ABB RobotStudio station: Tp1_20201210-163829.rsstn

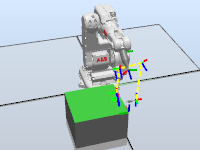
Station Tp1 (saved by RobotStudio 20.2.9116.0)
Controller IRB_140_6kg_0.81m
  mechanical unit ROB_1: IRB140_6_81_C_03, 6 joints, base frame (0, 0, 0) mm
Layout (positions relative to the parent item):
  - IRB140_6_81_C_03 [mechanism, from Robots\IRB140_6_81_C_G_03.rslib] at (0, 0, 0) mm; joint values [0, 0, 0, 3.1416, -0.5236, 3.1416] (rad or m)
  - Mesa [part]
  - Perno [part] at (0, 0, 0) mm
  - Pinza [mechanism] at (506.29, 0, 679.5) mm, rotated rx -180 ry 60 rz -180 deg
      TCP Pinza at (0, 0, 137) mm, rotated rx 0 ry 0 rz -22.5 deg
      links: Dummy
Attachment: Pinza is attached to IRB140_6_81_C_03 / Link6
EventTableEntry 1017: Group=, Trigger=DO_Pinza 1018, Actions=[EventTableActionAttach 1019], Comment=, ActivationMode=2, Cyclic=false
EventTableTriggerIO 1018: IOValue=[1], IRC5Controller=? -1, Operator=0, SignalSource=IRB_140_6kg_0.81m 515
EventTableActionAttach 1019: AttachmentParent=Pinza 1013, AttachmentChild=Perno 1009, MountObject=false, Offset=[X=1, Y=0, Z=0, W=0, X=0, Y=1, Z=0, W=0, X=0, Y=0, Z=1, W=0, X=0, Y=0, Z=0, W=1], FlangeIndext=0, FindNearest=false
EventTableEntry 1020: Group=, Trigger=DO_Pinza 1021, Actions=[EventTableActionDetach 1022], Comment=, ActivationMode=2, Cyclic=false
EventTableTriggerIO 1021: IOValue=[0], IRC5Controller=? -1, Operator=0, SignalSource=IRB_140_6kg_0.81m 515
EventTableActionDetach 1022: AttachmentParent=Pinza 1013, AttachmentChild=Perno 1009
Collision set Colision Perno- Mesa: Perno against Mesa, near miss 0.02 m
Collision set Colision Robot - Mesa: IRB140_6_81_C_03 against Mesa, near miss 0 m
Collision set Colision Pinza - Mesa: Mesa against Pinza, near miss 0 m
EventTableTriggerIO 1093: IOValue=[1], IRC5Controller=? -1, Operator=0, SignalSource=IRB_140_6kg_0.81m 515
EventTableTriggerIO 1094: IOValue=[0], IRC5Controller=? -1, Operator=0, SignalSource=IRB_140_6kg_0.81m 515
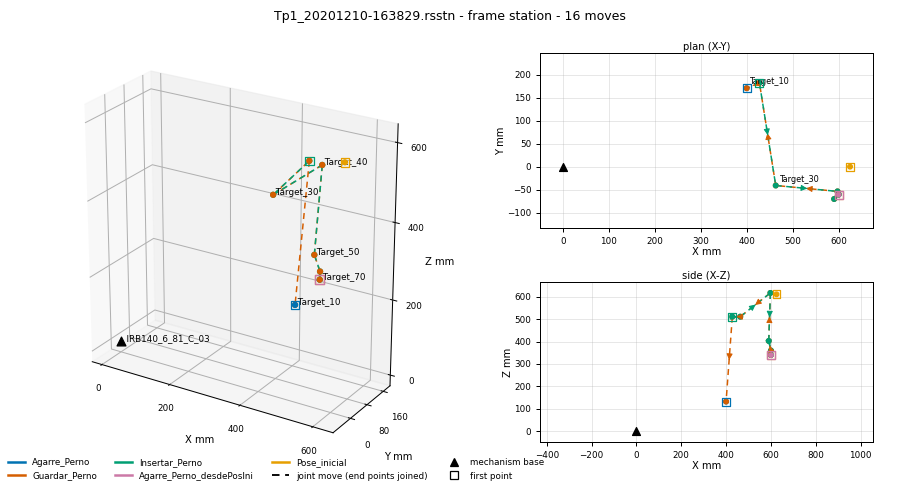
[picture p0: tool path of Tp1_20201210-163829.rsstn in frame station, 16 of 16 moves have a stored position in this frame; points joined in program order, loops and branches not executed]
Targets, tools, work objects and paths stored in the station, written as RAPID:
! task T_ROB1
MODULE CalibData
  PERS tooldata Pinza:=[TRUE,[[0,0,137],[0.98078528,0,0,-0.195090322]],[0.5,[0,0,100],[1,0,0,0],0,0,0]];
  PERS wobjdata wobjMesa:=[FALSE,TRUE,"",[[665,5,260],[0,0,0,1]],[[0,0,0],[1,0,0,0]]];
ENDMODULE

! task T_ROB1
MODULE Module1
  CONST robtarget PosicionInicial:=[[40.062869907,5,350.999997451],[0.09754516,-0.849384972,-0.168953176,0.490392634],[0,2,1,1],[9E+09,9E+09,9E+09,9E+09,9E+09,9E+09]];
  CONST robtarget PosicionInicial_:=[[624.937130551,0.000010862,610.999988852],[0.490392593,-0.168953224,0.849384987,-0.097545151],[0,2,1,1],[9E+09,9E+09,9E+09,9E+09,9E+09,9E+09]];
  CONST robtarget AgarrarPerno_:=[[400,170,130],[1,0,0,0],[0,0,0,0],[9E+09,9E+09,9E+09,9E+09,9E+09,9E+09]];
  CONST robtarget Target_10:=[[399.876122575,170.7866443,132.337906114],[0.008912565,-0.719405011,-0.69453365,0.000069399],[0,2,3,1],[9E+09,9E+09,9E+09,9E+09,9E+09,9E+09]];
  CONST robtarget Target_20:=[[427.713987214,182.423825838,511.144112895],[0.15413691,0.642318474,0.625246262,0.415615089],[0,2,3,1],[9E+09,9E+09,9E+09,9E+09,9E+09,9E+09]];
  CONST robtarget Target_30:=[[463.185948976,-40.945061339,511.144101517],[0.250584969,0.775091328,0.450265835,0.365651863],[-1,2,3,1],[9E+09,9E+09,9E+09,9E+09,9E+09,9E+09]];
  CONST robtarget Target_40:=[[597.654187124,-53.807206193,617.157465429],[0.010939233,0.861463336,-0.047210077,0.505502189],[-1,2,4,1],[9E+09,9E+09,9E+09,9E+09,9E+09,9E+09]];
  CONST robtarget Target_50:=[[590.340605336,-70.349210278,402.927571231],[0.041348347,0.698419889,-0.07410817,0.710639115],[-1,2,4,0],[9E+09,9E+09,9E+09,9E+09,9E+09,9E+09]];
  CONST robtarget Target_60:=[[600.000026092,-60.000012764,359.999989525],[0.041443001,0.709709838,-0.074523715,0.699314407],[-1,2,4,0],[9E+09,9E+09,9E+09,9E+09,9E+09,9E+09]];
  CONST robtarget Target_70:=[[600.000030476,-60.999977936,340.000067673],[0.041443276,0.709709587,-0.074523192,0.699314701],[-1,2,4,0],[9E+09,9E+09,9E+09,9E+09,9E+09,9E+09]];
  PROC Agarre_Perno()
    MoveJ Target_10,v100,fine,Pinza\WObj:=wobj0;
  ENDPROC
  PROC main()
    Pose_inicial;
    Agarre_Perno;
    SetDO DO_Pinza,1;
    Insertar_Perno;
    SetDO DO_Pinza,0;
    Pose_inicial;
    WaitTime 2;
    Agarre_Perno_desdePosInicial;
    SetDO DO_Pinza,1;
    Guardar_Perno;
    SetDO DO_Pinza,0;
    Pose_inicial;
  ENDPROC
  PROC Guardar_Perno()
    MoveJ Target_70,v500,fine,Pinza\WObj:=wobj0;
    MoveJ Target_60,v500,fine,Pinza\WObj:=wobj0;
    MoveJ Target_50,v500,fine,Pinza\WObj:=wobj0;
    MoveJ Target_40,v500,fine,Pinza\WObj:=wobj0;
    MoveJ Target_30,v500,fine,Pinza\WObj:=wobj0;
    MoveJ Target_20,v500,fine,Pinza\WObj:=wobj0;
    MoveJ Target_10,v500,fine,Pinza\WObj:=wobj0;
  ENDPROC
  PROC Insertar_Perno()
    MoveJ Target_20,v100,fine,Pinza\WObj:=wobj0;
    MoveJ Target_30,v100,fine,Pinza\WObj:=wobj0;
    MoveJ Target_40,v100,fine,Pinza\WObj:=wobj0;
    MoveJ Target_50,v100,fine,Pinza\WObj:=wobj0;
    MoveJ Target_60,v100,fine,Pinza\WObj:=wobj0;
    MoveJ Target_70,v100,fine,Pinza\WObj:=wobj0;
  ENDPROC
  PROC Agarre_Perno_desdePosInicial()
    MoveJ Target_70,v1000,fine,Pinza\WObj:=wobj0;
  ENDPROC
  PROC Pose_inicial()
    MoveJ PosicionInicial,v1000,z100,Pinza\WObj:=wobjMesa;
  ENDPROC
ENDMODULE

